# EPICS substitutions: ek9000App/Db/EL1808_mbbiDirect.substitutions
file EL1808.template
{       pattern
        {
                TERMINAL,

        }
        {
        }
}
